{attribute 'qualified_only'}
TYPE E_StationState :
(
	eAuto	:= 0,
	eManual := 1,
	eStop	:= 2	
);
END_TYPE

(* stored: Version 1.1.0.1, ProductVersion 3.1.4022.10
   DUT E_StationState: Id {c4de5c8d-c9b8-459b-b20e-9612fe2b2b83} *)
